{attribute addProperty BoxType "EL5101--0000"}
{attribute addProperty Id "Channel_1AT %I*Channel_6F37F4E44050Channel_1_1AT %Q*Channel_4D4E89362430WcStateAT %I*WcState_F855686C1620InfoDataAT %I*InfoData_BC63D37F80100"}
{attribute addProperty CRC "770969582"}
{attribute addProperty SizeInBites "160"}
{attribute addProperty SizeInBytes "20"}
TYPE EL5101_4D0D82F5 :
STRUCT
	{attribute addProperty Name "Channel_1"}
	Channel_1 : Channel_6F37F4E4;
	{attribute addProperty Name "Channel_1_1"}
	Channel_1_1 : Channel_4D4E8936;
	{attribute addProperty Name "WcState"}
	WcState : WcState_F855686C;
	{attribute addProperty Name "InfoData"}
	InfoData : InfoData_BC63D37F;
END_STRUCT
END_TYPE

(* stored: Version 1.2.0.0, ProductVersion 3.1.4024.9
   DUT EL5101_4D0D82F5: Id {025bad9d-59d4-43dd-a2f7-a17cb7291c1c} *)
